TYPE ST_SectorsConfig :
STRUCT
	AllSectorsConfig : REFERENCE TO ARRAY[GC.MIN_SECTOR_CT..GC.MAX_SECTOR_CT] OF ST_SectorConfig;
END_STRUCT
END_TYPE

(* stored: Version 1.1.0.1
   DUT ST_SectorsConfig: Id {f176946b-7df8-43f0-a166-08d19b370e57} *)
